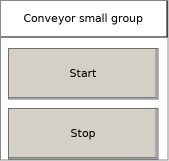
VISUALIZATION Frame_ConveyorSmallGroup  // 169x161
VAR_IN_OUT
	vio_fbConveyor1 : FB_Conveyor;
	vio_fbConveyor2 : FB_Conveyor;
	vio_fbConveyor3 : FB_Conveyor;
	vio_fbConveyor4 : FB_Conveyor;
END_VAR
    Button (8,48 150x51), "Start"
        OnMouseDown: execute {
            vio_fbConveyor1.in_bStart := TRUE;
            vio_fbConveyor2.in_bStart := TRUE;
            vio_fbConveyor3.in_bStart := TRUE;
            vio_fbConveyor4.in_bStart := TRUE;
        }
    Button (8,108 150x51), "Stop"
        OnMouseDown: execute {
            vio_fbConveyor1.in_bStop := TRUE;
            vio_fbConveyor2.in_bStop := TRUE;
            vio_fbConveyor3.in_bStop := TRUE;
            vio_fbConveyor4.in_bStop := TRUE;
        }
    Rectangle (0,0 167x37), "Conveyor small group"
END_VISUALIZATION

(* stored: Version 1.1.0.1, ProductVersion 3.1.4022.16
   Visu Frame_ConveyorSmallGroup: Id {63037a48-8368-4dd9-aa89-f5f66aa6e8ee} *)
